// SIMATIC S7-200 project (STEP 7-Micro/WIN), CPU 224 REL 02.01

SYMBOL_TABLE USUARIO1
PRESELECCION     I0.0
EJECUCION        I0.1
EMERGENCIA       I0.2
S0               I0.3
S1               I0.4
S2               I0.5
S3               I0.6
S4               I0.7
S5               I1.0
MEZCLA_1         Q0.0
MEZCLA_2         Q0.1
MEZCLA_3         Q0.2
MEZCLA_4         Q0.3
MEZCLA_5         Q0.4
MEZCLA_6         Q0.5
VALVULA_A        Q0.6
VALVULA_B        Q0.7
VALVULA_C        Q1.0
HOMOGENIZADOR    Q1.1
END_SYMBOL_TABLE

ORGANIZATION_BLOCK PRINCIPAL:OB1
TITLE=COMENTARIOS DEL PROGRAMA
BEGIN
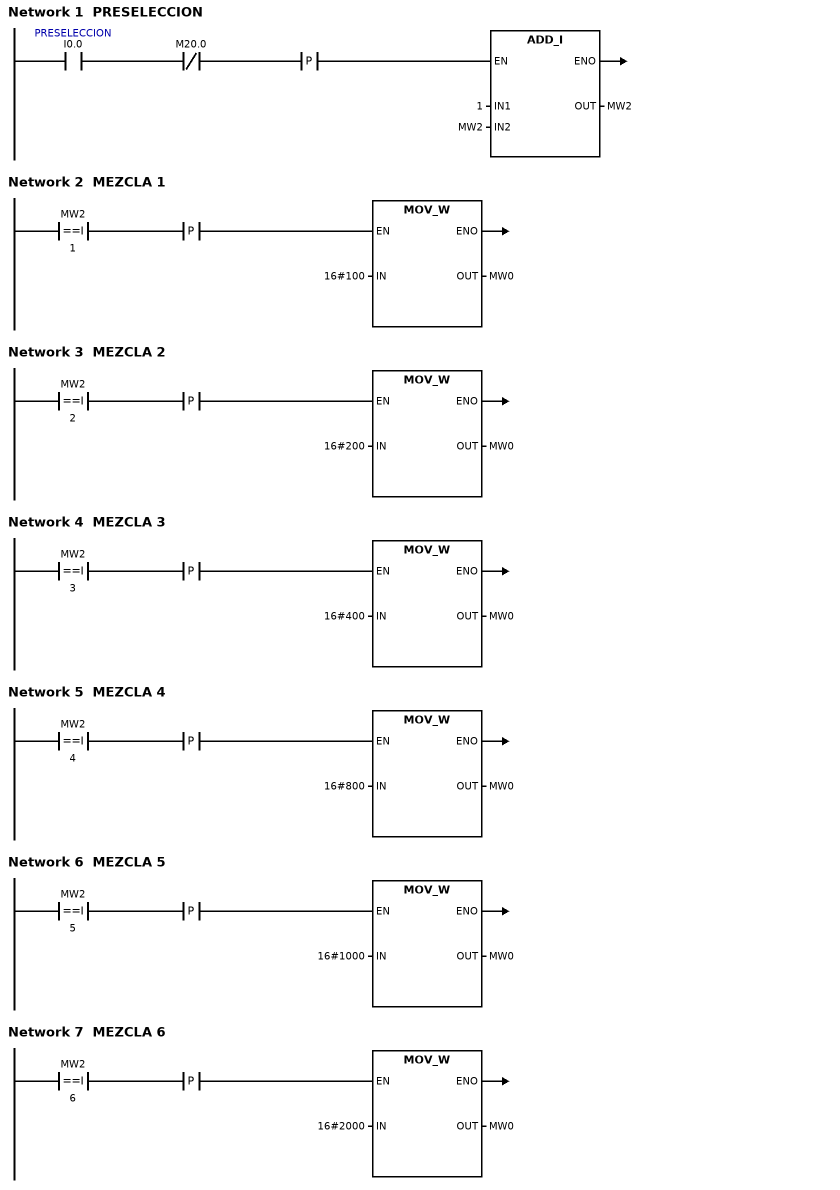
Network 1 // PRESELECCION
LD     PRESELECCION:I0.0
AN     M20.0
EU
+I     1, MW2
Network 2 // MEZCLA 1 
LDW=   MW2, 1
EU
MOVW   16#100, MW0
Network 3 // MEZCLA 2 
LDW=   MW2, 2
EU
MOVW   16#200, MW0
Network 4 // MEZCLA 3 
LDW=   MW2, 3
EU
MOVW   16#400, MW0
Network 5 // MEZCLA 4 
LDW=   MW2, 4
EU
MOVW   16#800, MW0
Network 6 // MEZCLA 5 
LDW=   MW2, 5
EU
MOVW   16#1000, MW0
Network 7 // MEZCLA 6 
LDW=   MW2, 6
EU
MOVW   16#2000, MW0
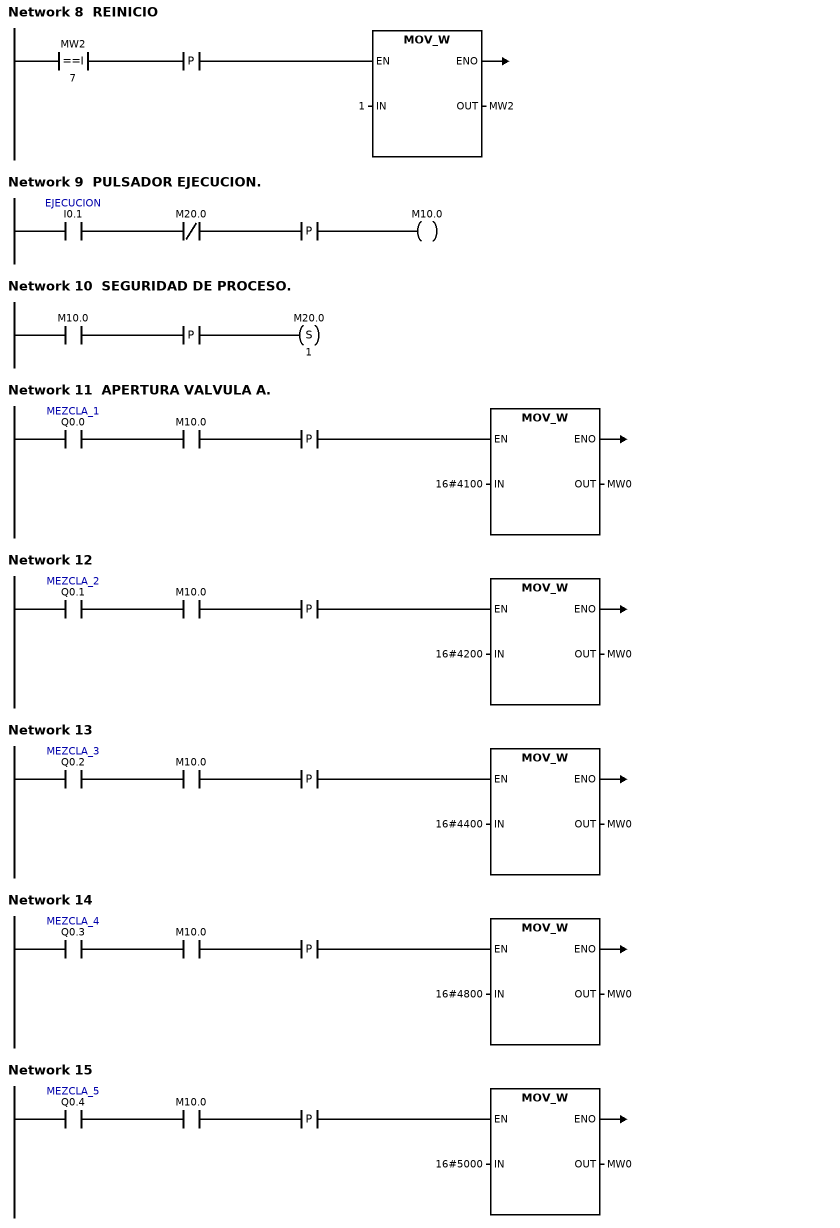
Network 8 // REINICIO
LDW=   MW2, 7
EU
MOVW   1, MW2
Network 9 // PULSADOR EJECUCION.
LD     EJECUCION:I0.1
AN     M20.0
EU
=      M10.0
Network 10 // SEGURIDAD DE PROCESO.
LD     M10.0
EU
S      M20.0, 1
Network 11 // APERTURA VALVULA A.
LD     MEZCLA_1:Q0.0
A      M10.0
EU
MOVW   16#4100, MW0
Network 12
LD     MEZCLA_2:Q0.1
A      M10.0
EU
MOVW   16#4200, MW0
Network 13
LD     MEZCLA_3:Q0.2
A      M10.0
EU
MOVW   16#4400, MW0
Network 14
LD     MEZCLA_4:Q0.3
A      M10.0
EU
MOVW   16#4800, MW0
Network 15
LD     MEZCLA_5:Q0.4
A      M10.0
EU
MOVW   16#5000, MW0
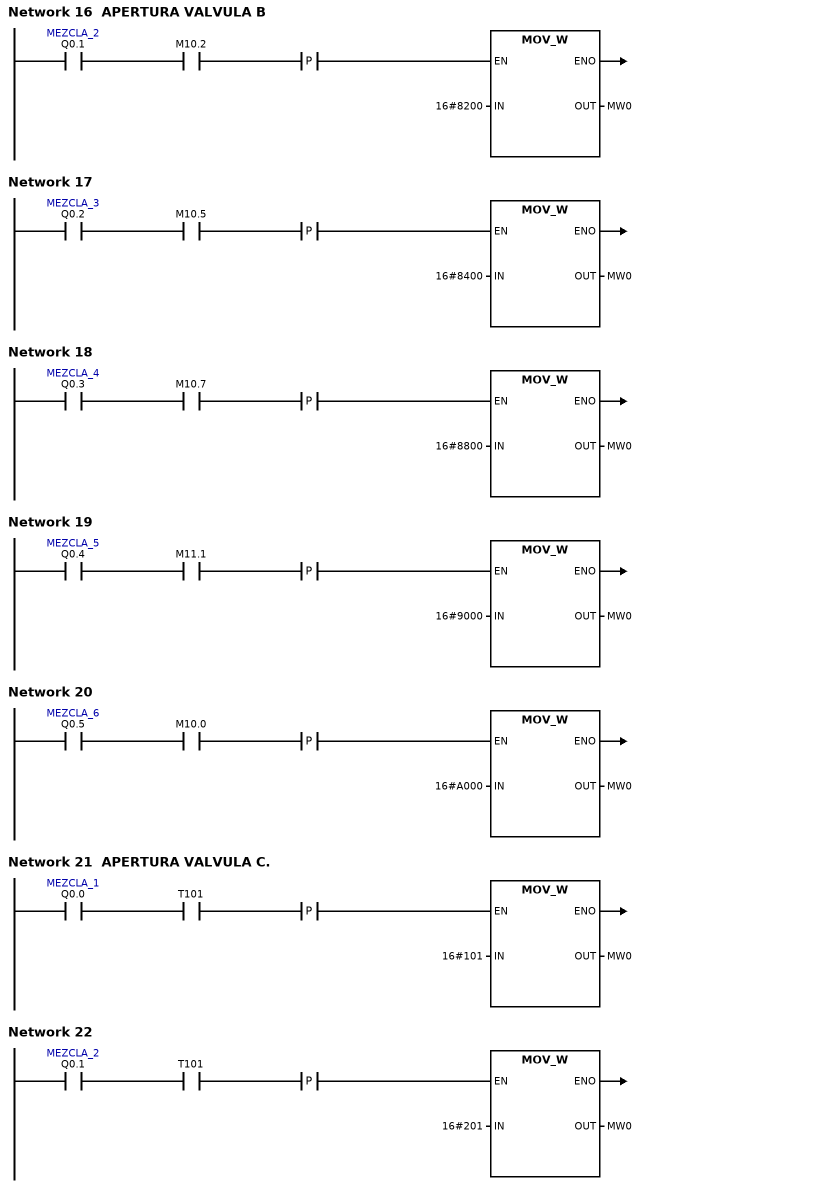
Network 16 // APERTURA VALVULA B
LD     MEZCLA_2:Q0.1
A      M10.2
EU
MOVW   16#8200, MW0
Network 17
LD     MEZCLA_3:Q0.2
A      M10.5
EU
MOVW   16#8400, MW0
Network 18
LD     MEZCLA_4:Q0.3
A      M10.7
EU
MOVW   16#8800, MW0
Network 19
LD     MEZCLA_5:Q0.4
A      M11.1
EU
MOVW   16#9000, MW0
Network 20
LD     MEZCLA_6:Q0.5
A      M10.0
EU
MOVW   16#A000, MW0
Network 21 // APERTURA VALVULA C.
LD     MEZCLA_1:Q0.0
A      T101
EU
MOVW   16#101, MW0
Network 22
LD     MEZCLA_2:Q0.1
A      T101
EU
MOVW   16#201, MW0
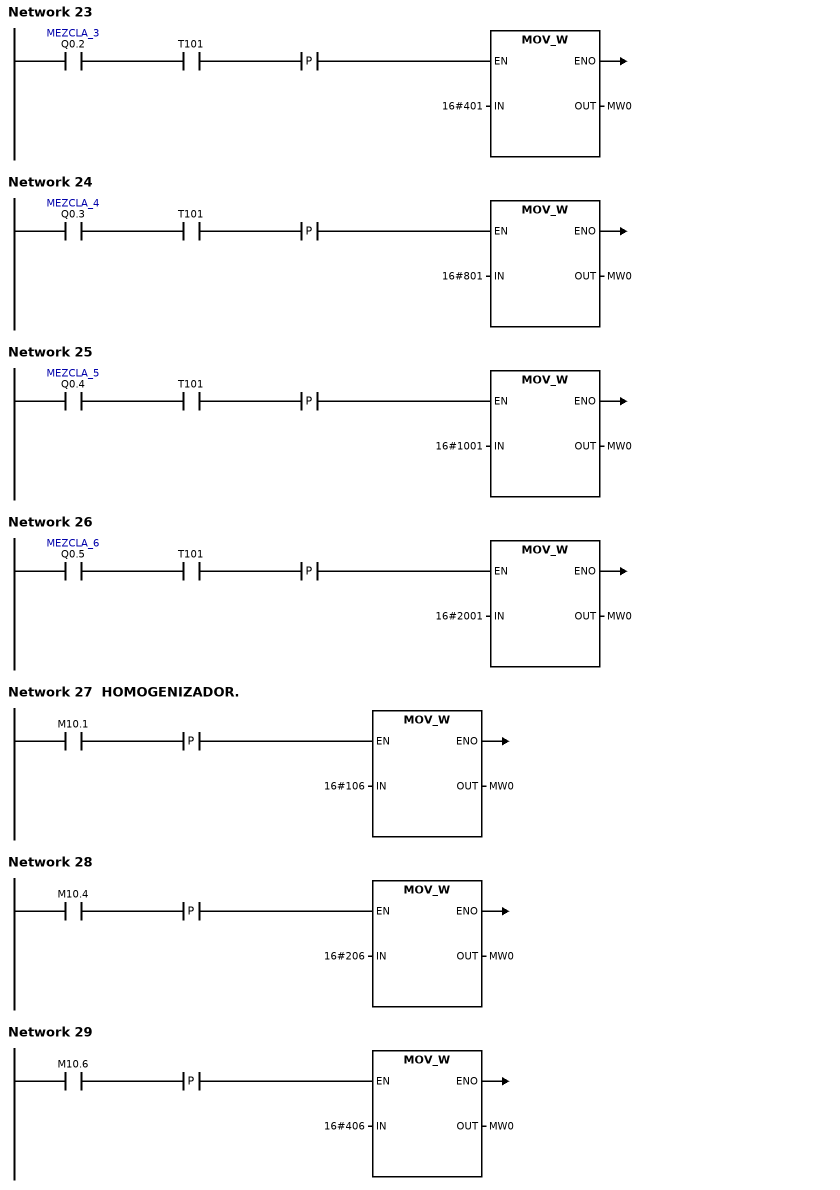
Network 23
LD     MEZCLA_3:Q0.2
A      T101
EU
MOVW   16#401, MW0
Network 24
LD     MEZCLA_4:Q0.3
A      T101
EU
MOVW   16#801, MW0
Network 25
LD     MEZCLA_5:Q0.4
A      T101
EU
MOVW   16#1001, MW0
Network 26
LD     MEZCLA_6:Q0.5
A      T101
EU
MOVW   16#2001, MW0
Network 27 // HOMOGENIZADOR.
LD     M10.1
EU
MOVW   16#106, MW0
Network 28
LD     M10.4
EU
MOVW   16#206, MW0
Network 29
LD     M10.6
EU
MOVW   16#406, MW0
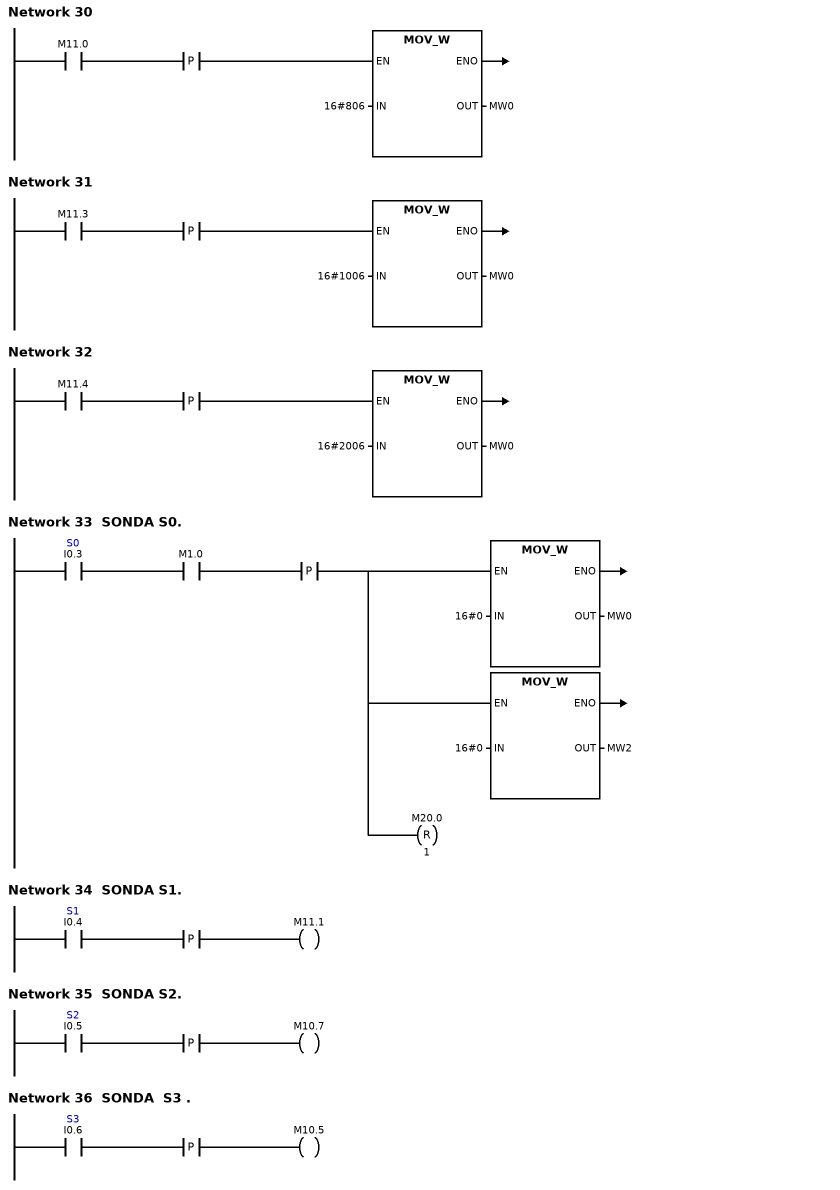
Network 30
LD     M11.0
EU
MOVW   16#806, MW0
Network 31
LD     M11.3
EU
MOVW   16#1006, MW0
Network 32
LD     M11.4
EU
MOVW   16#2006, MW0
Network 33 // SONDA S0.
LD     S0:I0.3
A      M1.0
EU
MOVW   16#0, MW0
MOVW   16#0, MW2
R      M20.0, 1
Network 34 // SONDA S1.
LD     S1:I0.4
EU
=      M11.1
Network 35 // SONDA S2.
LD     S2:I0.5
EU
=      M10.7
Network 36 // SONDA  S3 .
LD     S3:I0.6
EU
=      M10.5
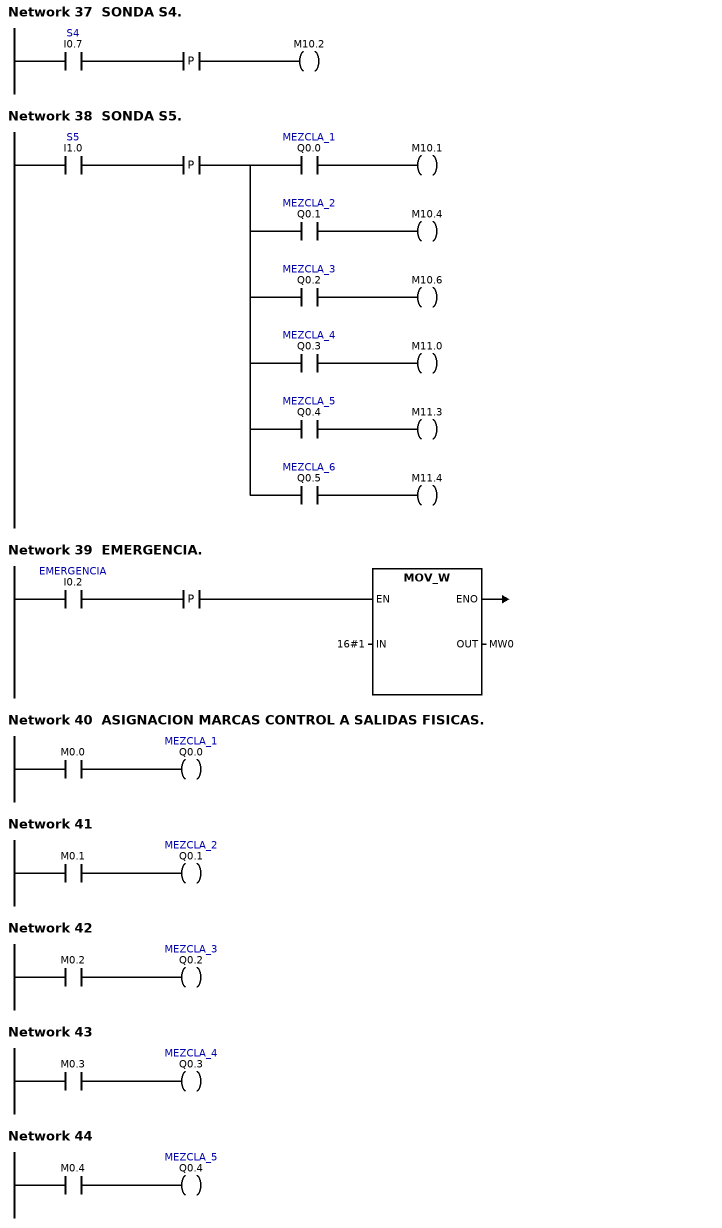
Network 37 // SONDA S4.
LD     S4:I0.7
EU
=      M10.2
Network 38 // SONDA S5.
LD     S5:I1.0
EU
LPS
A      MEZCLA_1:Q0.0
=      M10.1
LRD
A      MEZCLA_2:Q0.1
=      M10.4
LRD
A      MEZCLA_3:Q0.2
=      M10.6
LRD
A      MEZCLA_4:Q0.3
=      M11.0
LRD
A      MEZCLA_5:Q0.4
=      M11.3
LPP
A      MEZCLA_6:Q0.5
=      M11.4
Network 39 // EMERGENCIA.
LD     EMERGENCIA:I0.2
EU
MOVW   16#1, MW0
Network 40 // ASIGNACION MARCAS CONTROL A SALIDAS FISICAS.
LD     M0.0
=      MEZCLA_1:Q0.0
Network 41
LD     M0.1
=      MEZCLA_2:Q0.1
Network 42
LD     M0.2
=      MEZCLA_3:Q0.2
Network 43
LD     M0.3
=      MEZCLA_4:Q0.3
Network 44
LD     M0.4
=      MEZCLA_5:Q0.4
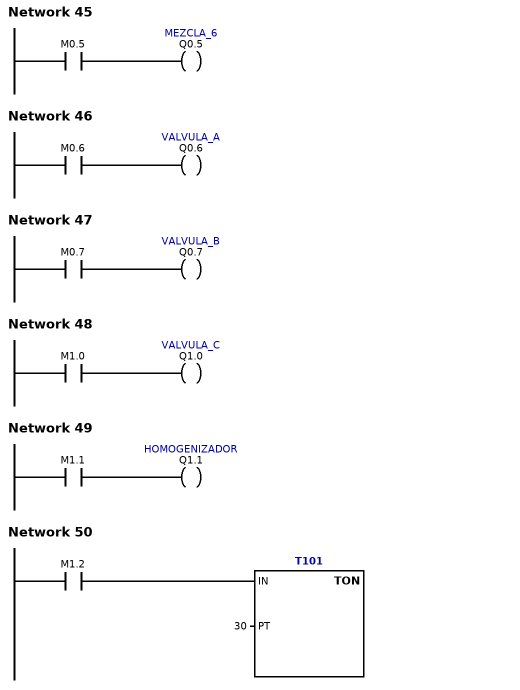
Network 45
LD     M0.5
=      MEZCLA_6:Q0.5
Network 46
LD     M0.6
=      VALVULA_A:Q0.6
Network 47
LD     M0.7
=      VALVULA_B:Q0.7
Network 48
LD     M1.0
=      VALVULA_C:Q1.0
Network 49
LD     M1.1
=      HOMOGENIZADOR:Q1.1
Network 50
LD     M1.2
TON    T101, 30
END_ORGANIZATION_BLOCK
